Staubli VAL3: POINT.pjx

--- POINT.pjx ---
Parameters version=s7.7 stackSize=5000 millimeterUnit=true
Program file=computeFrame.pgx
Program file=delete.pgx
Program file=deleteItem.pgx
Program file=duplicate.pgx
Program file=find.pgx
Program file=get.pgx
Program file=getDistance.pgx
Program file=getFrame.pgx
Program file=getFrameId.pgx
Program file=getFunctionEdit.pgx
Program file=getFunctionSel.pgx
Program file=getFunctionView.pgx
Program file=getListItem.pgx
Program file=getPoint.pgx
Program file=getSize.pgx
Program file=getSizeItem.pgx
Program file=getTime.pgx
Program file=getTool.pgx
Program file=getTrajItem.pgx
Program file=getTrajType.pgx
Program file=getType.pgx
Program file=goTo.pgx
Program file=HerePoint.pgx
Program file=insertItem.pgx
Program file=load.pgx
Program file=loadCycle.pgx
Program file=loadPage.pgx
Program file=makeTraj.pgx
Program file=new.pgx
Program file=onEdit.pgx
Program file=onEditItem.pgx
Program file=onEditTrsf.pgx
Program file=onFunctionEdit.pgx
Program file=onFunctionSel.pgx
Program file=onFunctionView.pgx
Program file=onInsert.pgx
Program file=onProgEnd.pgx
Program file=onRun.pgx
Program file=onSave.pgx
Program file=onStart.pgx
Program file=onStop.pgx
Program file=setFrameId.pgx
Program file=setTool.pgx
Program file=setTrajItem.pgx
Data file=POINT.dtx
Library alias=saveData path=Disk://saveData/saveData.pjx
Library alias=page path=Disk://kernel/template/page/page.pjx
Library alias=use path=Disk://kernel/userPage/userPage.pjx
Library alias=language path=Disk://kernel/language/language.pjx
Library alias=tcp path=Disk://kernel/tool/tool.pjx
Library alias=cycleStatus path=Disk://cycleStatus/cycleStatus.pjx
Library alias=pt path=Disk://kernel/template/session/saveTraj/POINT/POINT.pjx
Type name=TrajectoryItem path=Disk://kernel/template/TrajectoryItem/TrajectoryItem.pjx
Type name=ActionItem path=Disk://kernel/template/ActionItem/ActionItem.pjx
Type name=Trajectory path=Disk://kernel/template/Trajectory/Trajectory.pjx
Type name=TrajPoint path=Disk://kernel/template/TrajPoint/TrajPoint.pjx
Type name=InstrItem path=Disk://kernel/template/InstrItem/InstrItem.pjx
Type name=FrameItem path=Disk://kernel/template/FrameItem/FrameItem.pjx
Type name=TrajPointItem path=Disk://kernel/template/TrajPointItem/TrajPointItem.pjx

--- POINT.dtx ---
Trajectory tTraj
  [0]
    TrajectoryItem tSuper[3]
      [0]
        num distance
        num moveType = 1
        num nTime
        num nStop
        num nTcpAction
        string comment = "appro"
        bool toStop
        mdesc nom_speed = {tmax=300, rmax=9999, leave=30, reach=30}
        InstrItem iInstr[3]
          [0]
            string sType
            string sData
          [1]
            string sType
            string sData
          [2]
            string sType
            string sData
        num nMoveId
      [1]
        num distance = 2
        num moveType = 1
        num nTime
        num nStop
        num nTcpAction = 2
        string comment = "point"
        bool toStop = true
        mdesc nom_speed = {tmax=300, rmax=9999, leave=30, reach=30}
        InstrItem iInstr[3]
          [0]
            string sType
            string sData
          [1]
            string sType
            string sData
          [2]
            string sType
            string sData
        num nMoveId
      [2]
        num distance
        num moveType = 1
        num nTime
        num nStop
        num nTcpAction
        string comment = "depart"
        bool toStop
        mdesc nom_speed = {tmax=300, rmax=9999, leave=30, reach=30}
        InstrItem iInstr[3]
          [0]
            string sType
            string sData
          [1]
            string sType
            string sData
          [2]
            string sType
            string sData
        num nMoveId
    string sID = "POINT pose"
    num nId
public bool bMoveType[3]
  [0] = true
  [1] = true
public bool bStepping
bool bToSave
frame fSetFrame = {fatherId=world[0]}
mdesc mMdesc = {accel=10, vel=10, decel=10, blend=off}
string sInstruction
public string sItems
string sMenu[8]
  [5] = "Duplicate"
  [7] = "New"
string sTrajType = "POINT"
pointRx pToGo = {fatherId=world[0]}
frame fFather = {fatherId=world[0]}
string sItemCycle
TrajPoint pEditPoint
  [0]
    TrajPointItem tData[3]
      [0]
        TrajectoryItem tSuper
          [0]
            num distance
            num moveType
            num nTime
            num nStop
            num nTcpAction
            string comment
            bool toStop
            mdesc nom_speed = {vel=500, tmax=500, rmax=9999, leave=30, reach=30}
            InstrItem iInstr[3]
              [0]
                string sType
                string sData
              [1]
                string sType
                string sData
              [2]
                string sType
                string sData
            num nMoveId
        pointRx pPoint = {fatherId=pEditPoint[0].fFrame[0]}
        num nType
      [1]
        TrajectoryItem tSuper
          [0]
            num distance
            num moveType
            num nTime
            num nStop
            num nTcpAction
            string comment
            bool toStop
            mdesc nom_speed = {vel=500, tmax=500, rmax=9999, leave=30, reach=30}
            InstrItem iInstr[3]
              [0]
                string sType
                string sData
              [1]
                string sType
                string sData
              [2]
                string sType
                string sData
            num nMoveId
        pointRx pPoint = {fatherId=pEditPoint[0].fFrame[0]}
        num nType
      [2]
        TrajectoryItem tSuper
          [0]
            num distance
            num moveType
            num nTime
            num nStop
            num nTcpAction
            string comment
            bool toStop
            mdesc nom_speed = {vel=500, tmax=500, rmax=9999, leave=30, reach=30}
            InstrItem iInstr[3]
              [0]
                string sType
                string sData
              [1]
                string sType
                string sData
              [2]
                string sType
                string sData
            num nMoveId
        pointRx pPoint = {fatherId=pEditPoint[0].fFrame[0]}
        num nType
    frame fFrame = {fatherId=world[0]}
    num nIndexTool
    string sID
    num nIndexFrame

--- computeFrame.pgx ---
public program computeFrame(num x_nNewFrame)
  local num i
begin
  // recompute all the point into the new frame
  for i=0 to size(pEditPoint.tData)-1
    if pEditPoint.tData[i].nType==1
      pEditPoint.tData[i].pPoint.trsf=position(pEditPoint.tData[i].pPoint,saveData:fFrameItem[x_nNewFrame].fFrame)
    endIf
  endFor
end

--- delete.pgx ---
public program delete(string x_sName (dimensions=1), num& x_nResult[] (dimensions=1))
  local string l_sItem
  local num l_nSize
begin
  //
  // delete the select trajectory
  //
  if isDefined(pt:tTraj[x_sName])
    // delete
    delete(pt:tTraj[x_sName])
    // save it
    bToSave=true
    x_nResult=0
  else
    x_nResult=-1
  endIf

end

--- deleteItem.pgx ---
public program deleteItem(num& x_nIndex (dimensions=1))
  local num i
  local string l_sItem
begin
  // delete the selected item
  if pEditPoint.tData[x_nIndex].nType!=1 and size(pEditPoint.tData)>3
    // delete all the field
    delete(pEditPoint.tData[x_nIndex])
  else
    // not possible to delete the point
    if pEditPoint.tData[x_nIndex].nType!=1
      pEditPoint.tData[x_nIndex].pPoint.trsf={0,0,0,0,0,0}
    endIf
    x_nIndex=-1
  endIf
end

--- find.pgx ---
public program find(string& x_sItem[] (dimensions=1), bool& x_bFound[] (dimensions=1))
begin
  // check if the item has been found
  x_bFound=isDefined(pt:tTraj[x_sItem])
end

--- get.pgx ---
public program get(string& x_sItem[] (dimensions=1), num x_nIndex (dimensions=1))
  local string l_sKey
  local num i
  local string l_sItem
begin
  // start from the first
  l_sKey=first(pt:tTraj)
  // search it
  while l_sKey!=""
    x_sItem=l_sKey
    l_sKey=next(pt:tTraj[l_sKey])
    if i==x_nIndex
      return
    else
      i=i+1
    endIf
  endWhile
end

--- getDistance.pgx ---
public program getDistance(tool x_tTool, num& x_nDistance[], bool x_bCycle, num x_nIndex)
  local point l_pPoint
  local num l_nValue
  local trsf l_trsfEmpty
  local point l_pActual
  local point l_pPrev
begin
  // first point
  if x_nIndex==0
    x_nDistance=10
    return
  else
    //
    // get the point
    //
    call getPoint(l_pActual,x_bCycle,x_nIndex)
    call getPoint(l_pPrev,x_bCycle,x_nIndex-1)
    if x_bCycle
      // an other one

      switch pt:tTraj[sItemCycle].tData[x_nIndex].nType
        case 0
          // appro
          x_nDistance=distance(position(l_pPrev,world),position(l_pActual,world))
        break
        case 1
          // point
          x_nDistance=distance(l_pPrev.trsf,l_trsfEmpty)
        break
        case 2
          // depart
          if pt:tTraj[sItemCycle].tData[x_nIndex-1].nType==1
            x_nDistance=distance(l_trsfEmpty,l_pActual.trsf)
          else
            x_nDistance=distance(position(l_pPrev,world),position(l_pActual,world))
          endIf
        break
      endSwitch
    else
      // an other one
      switch pEditPoint[x_nIndex].tData.nType
        case 0
          // appro
          x_nDistance=distance(position(l_pPrev,world),position(l_pActual,world))
        break
        case 1
          // point
          x_nDistance=distance(l_pPrev.trsf,l_trsfEmpty)
        break
        case 2
          // depart
          if pEditPoint[x_nIndex-1].tData.nType==1
            x_nDistance=distance(l_trsfEmpty,l_pActual.trsf)
          else
            x_nDistance=distance(position(l_pPrev,world),position(l_pActual,world))
          endIf
        break
      endSwitch
    endIf
  endIf
end

--- getFrame.pgx ---
public program getFrame(frame& x_fFrame[], bool x_bCycle)
begin
  if x_bCycle
    x_fFrame.trsf=position(pt:tTraj[sItemCycle].fFrame,world)
  else
    // update the frame
    x_fFrame.trsf=position(pEditPoint.fFrame,world)
  endIf
end

--- getFrameId.pgx ---
public program getFrameId(num& x_nFrame)
begin
  // give back the frame
  x_nFrame=pEditPoint.nIndexFrame
end

--- getFunctionSel.pgx ---
public program getFunctionSel(string& x_sName[] (dimensions=1))
  local string l_sMessage
begin
  //
  // define your message for the
  // function KEY
  //
  // NOTE is an ARRAY[0..7]
  //
  // example:
  // x_sName[1]="DEMO"
  // active the F2 button
  //
end

--- getListItem.pgx ---
public program getListItem(string& x_sItem[] (dimensions=1), num x_nIndex (dimensions=1))
  local trsf l_tTrsf
  local string l_sItem[6]
  local string l_sEvent
begin
  //
  // define the item to show in the edit page Traj
  // customize an array and copy to x_sItem...
  //
  // see other traj as example
  // 0 > appro
  // 1 > point
  // 2 > depart
  // take it
  switch pEditPoint.tData[x_nIndex].nType
    case 0
      l_sEvent="appro  "
    break
    case 1
      l_sEvent="coord  "
    break
    case 2
      l_sEvent="depart "
    break
  endSwitch
  l_tTrsf=pEditPoint.tData[x_nIndex].pPoint.trsf
  // show them
  l_sItem[0]=(l_sEvent+" X > "+toString(".2",l_tTrsf.x))
  l_sItem[1]=(l_sEvent+" Y > "+toString(".2",l_tTrsf.y))
  l_sItem[2]=(l_sEvent+" Z > "+toString(".2",l_tTrsf.z))
  l_sItem[3]=(l_sEvent+"RX > "+toString(".2",l_tTrsf.rx))
  l_sItem[4]=(l_sEvent+"RY > "+toString(".2",l_tTrsf.ry))
  l_sItem[5]=(l_sEvent+"RZ > "+toString(".2",l_tTrsf.rz))
  // look for intermediate point
  call use:stringCopy(l_sItem,x_sItem)
end

--- getPoint.pgx ---
public program getPoint(point& x_pPoint[], bool x_bCycle, num x_nIndex)
  local string l_sItem
  local num l_nSize
  local num i
  local num l_nPoint
begin
  // take
  if x_bCycle
    // in Cycle
    switch pt:tTraj[sItemCycle].tData[x_nIndex].nType
      case 0,2
        call getSizeItem(true,l_nSize)
        for i=0 to l_nSize-1
          // scan for the real point
          if pt:tTraj[sItemCycle].tData[i].nType==1
            l_nPoint=i
            i=l_nSize-1
          endIf
        endFor
        // give back
        x_pPoint=appro(pt:tTraj[sItemCycle].tData[l_nPoint].pPoint,pt:tTraj[sItemCycle].tData[x_nIndex].pPoint.trsf)
      break
      case 1
        // real point
        x_pPoint=pt:tTraj[sItemCycle].tData[x_nIndex].pPoint
      break
    endSwitch
  else
    // not in Cycle
    switch pEditPoint.tData[x_nIndex].nType
      case 0,2
        call getSizeItem(false,l_nSize)
        for i=0 to l_nSize-1
          // scan for the real point
          if pEditPoint.tData[i].nType==1
            l_nPoint=i
            i=l_nSize-1
          endIf
        endFor
        // give back
        x_pPoint=appro(pEditPoint.tData[l_nPoint].pPoint,pEditPoint.tData[x_nIndex].pPoint.trsf)
      break
      case 1
        // real point
        x_pPoint=pEditPoint.tData[x_nIndex].pPoint
      break
    endSwitch
  endIf
end

--- getSize.pgx ---
public program getSize(num& x_nSize[] (dimensions=1))
  local string l_sType
  local string l_sKey
  local num i
  local string l_sItem
  local string l_sPath
  local num l_nResult
begin
  // give back the size
  x_nSize=size(pt:tTraj)
end

--- getSizeItem.pgx ---
public program getSizeItem(bool x_bCycle, num& x_nSize)
  local string l_sType
  local string l_sKey
  local num i
begin
  //
  // get the size of the collection
  //
  if x_bCycle
    x_nSize=size(pt:tTraj[sItemCycle].tData)
  else
    x_nSize=size(pEditPoint.tData)
  endIf
end

--- getTime.pgx ---
public program getTime(num& x_nTime[], bool x_bCycle, num x_nIndex)
begin
  // get the time DATA
  if x_bCycle
    // get the time DATA
    x_nTime=pt:tTraj[sItemCycle].tData[x_nIndex].tSuper.nTime
  else
    // get the time DATA
    x_nTime=pEditPoint.tData[x_nIndex].tSuper.nTime
  endIf
end

--- getTool.pgx ---
public program getTool(num& x_nTool (dimensions=1))
begin
  // edit one
  x_nTool=pEditPoint.nIndexTool
end

--- getTrajItem.pgx ---
public program getTrajItem(TrajectoryItem& x_tTraj[] (dimensions=1), num x_nIndex (dimensions=1))
begin
  //
  // get all the FIELD
  //
  x_tTraj=pEditPoint.tData[x_nIndex].tSuper
end

--- getTrajType.pgx ---
program getTrajType(string& x_sTrajType[] (dimensions=1))
  local num l_nPos
  local string l_sPath
begin
  // get the trajType
  l_sPath=libPath()
  if find(l_sPath,sTrajType)==-1 or sTrajType==""
    do
      l_nPos=find(l_sPath,"/")
      if l_nPos==-1
        l_nPos=find(l_sPath,"\")
      endIf
      if l_nPos!=-1
        l_sPath=right(l_sPath,len(l_sPath)-l_nPos-1)
      endIf
    until l_nPos==-1
    //
    sTrajType=l_sPath
  endIf
  // return back
  x_sTrajType=sTrajType
end

--- getType.pgx ---
public program getType(num& x_nType, bool x_bCycle, num x_nIndex)
begin
  // get the point Type
  if x_bCycle
    x_nType=pt:tTraj[sItemCycle].tData[x_nIndex].nType
  else
    x_nType=pEditPoint.tData[x_nIndex].nType
  endIf
end

--- goTo.pgx ---
public program goTo(tool x_tTool, mdesc x_mDesc, num x_nMoveType, bool& x_bUnreached[], num x_nIndex)
  local point l_pTrsf
  local bool l_bInside
  local tool l_tTool
  local point l_pHere
  local string l_sMessage
  local num l_nSize
  local num i
  local mdesc l_mSpeed
  local joint l_jHere
  local joint l_jJoint
begin
  // the maximum size
  call getSizeItem(false,l_nSize)
  // get the trsf
  call getPoint(pToGo,false,x_nIndex)
  // check if the point is ok
  if pointToJoint(x_tTool,herej(),pToGo,l_jJoint)
    // step by step motion
    if x_nMoveType==0
      // or is not in range
      movej(pToGo,x_tTool,x_mDesc)
    else
      movel(pToGo,x_tTool,x_mDesc)
    endIf
  else
    // get the message point is not reachable
    call language:message(l_sMessage,-5)
    call use:type(0,12,"!!! "+l_sMessage)
  endIf
end

--- HerePoint.pgx ---
public program HerePoint(num x_nIndex)
  local tool l_tTool
  local point l_pHere
  local frame l_fFrame
  local num i
  local num l_nIndex
  local num l_nSize
  local string l_sMessage
begin
  //
  // take the point
  //
  // frame
  call getFrame(fSetFrame,false)
  // tool
  call tcp:getTool(l_tTool,pEditPoint.nIndexTool)
  // here
  l_pHere=here(l_tTool,fSetFrame)
  resetMotion()
  // check the index
  if pEditPoint.tData[x_nIndex].nType==1
    // save the trsf
    pEditPoint.tData[x_nIndex].pPoint.trsf=l_pHere.trsf
  else
    // search for the index of the point
    call getSizeItem(false,l_nSize)
    for i=0 to l_nSize-1
      if pEditPoint.tData[i].nType==1
        // save and exit
        l_nIndex=i
        i=l_nSize
      endIf
    endFor
    if pEditPoint.tData[l_nIndex].pPoint.trsf!={0,0,0,0,0,0}
      // compute the approch
      pEditPoint.tData[x_nIndex].pPoint.trsf=!pEditPoint.tData[l_nIndex].pPoint.trsf*l_pHere.trsf
    else
      // point not taught
      call language:message(l_sMessage,147)
      popUpMsg(l_sMessage)
    endIf
  endIf
  // check the moveType to save the config
  if pEditPoint.tData[x_nIndex].tSuper.moveType==0
    pEditPoint.tData[x_nIndex].pPoint.config=l_pHere.config
  else
    pEditPoint.tData[x_nIndex].pPoint.config={ssame,esame,wfree}
  endIf
  // to be save

end

--- insertItem.pgx ---
public program insertItem(num& x_nIndexCopy, num x_nIndexPaste)
  local num l_nLastType
  local point l_pPoint
  local num l_nType
begin
  //
  // use to add more elements from the typical one
  //
  // insert all the field
  //
  l_pPoint=pEditPoint.tData[x_nIndexCopy].pPoint
  l_nLastType=pEditPoint.tData[x_nIndexCopy].nType
  if l_nLastType==0
    l_nType=0
  elseIf l_nLastType==2 or l_nLastType==1
    l_nType=2
  endIf
  insert(pEditPoint.tData[x_nIndexPaste])
  // set IT - link it
  link(pEditPoint.tData[x_nIndexPaste].pPoint,pEditPoint.fFrame)
  pEditPoint.tData[x_nIndexPaste].pPoint.trsf=l_pPoint.trsf
  // set IT
  pEditPoint.tData[x_nIndexPaste].nType=l_nType
end

--- load.pgx ---
public program load(string x_sItem, num& x_nResult)
  local string l_sType
  local string l_sMessage
  local num i
begin
  // load the select trajectory..already loaded
  call getTrajType(l_sType)
  if find(pt:libPath(),saveData:sPathTraj)==-1
    pt:libLoad(saveData:sPathTraj+l_sType)
      delay(0)
    if saveData:bDebug
      ? "loading POINT..."+saveData:sPathTraj+l_sType
    endIf
  endIf
  // use the type...
  if isDefined(pt:tTraj[x_sItem])
    // link the frame and all the points
    call pt:link_all(x_sItem)
    // check if link and defined
    pEditPoint=pt:tTraj[x_sItem]
    pEditPoint.sID=x_sItem
  elseIf x_sItem!=""
    // not FOUND
    call language:message(l_sMessage,-7)
    x_nResult=-1
    popUpMsg(l_sMessage+x_sItem)
  endIf
end

--- loadCycle.pgx ---
public program loadCycle(string x_sItem, num& x_nResult[])
  local string l_sType
  local string l_sMessage
begin
  // load the select trajectory..already loaded
  call getTrajType(l_sType)
  if find(pt:libPath(),saveData:sPathTraj)==-1
    pt:libLoad(saveData:sPathTraj+l_sType)
    delay(0)
    if saveData:bDebug
      ? "loading POINT..."+saveData:sPathTraj+l_sType
    endIf
  endIf
  if isDefined(pt:tTraj[x_sItem])
    // link the frame and all the points
    call pt:link_all(x_sItem)
    sItemCycle=x_sItem
  else
    // not FOUND
    call language:message(l_sMessage,-7)
    x_nResult=-1
    cycleStatus:bToStop=true
    popUpMsg(l_sMessage+x_sItem)
  endIf
end

--- loadPage.pgx ---
program loadPage(string x_sPage, string& x_sItems[])
// load the next page
  local num i
begin
  // look if the page libload is correct
  i=page:libLoad(x_sPage)
  delay(0)
  logMsg("KERNEL:PAGE LIBLOAD "+x_sPage+" result "+toString("",i))
  if i!=0
    popUpMsg("Loading page "+x_sPage+" error CODE "+toString("",i))
  else
    page:sItems=x_sItems
    call page:main()
  endIf
end

--- makeTraj.pgx ---
public program makeTraj(string& x_sItem[])
  local num i
  local num l_nDistance
  local num l_nSize
  local tool l_tTool
  local bool l_bToStop
  local mdesc l_mDesc
  local num l_nMoveId
  local bool l_bOk
  local string l_sType
  local TrajectoryItem l_tTraj
  local ActionItem l_aAction
  local point l_pPoint
begin
  // take the TOOL
  call tcp:getTool(l_tTool,pt:tTraj[sItemCycle].nIndexTool)
  // the maximum size
  call getSizeItem(true,l_nSize)
  //
  // for all of my traj cyclePoints move the robot
  //
  resize(tTraj.tSuper,1,size(pt:tTraj[sItemCycle].tData))
  for i=0 to (l_nSize-1)
    tTraj.tSuper[i]=pt:tTraj[sItemCycle].tData[i].tSuper
  endFor
  tTraj.sID="POINT "+pt:tTraj[sItemCycle].sID
  call cycleStatus:addTraj(tTraj)
  //
  // for all of my traj cyclePoints move the robot
  //
  for i=0 to (l_nSize-1)
    //
    // get the point info
    //
    l_tTraj=pt:tTraj[sItemCycle].tData[i].tSuper
    call getPoint(l_pPoint,true,i)
    //
    // get the distance in percentage
    call getDistance(l_tTool,l_nDistance,true,i)
    //
    // give to the traj library the percentage distance
    //
    if l_bToStop
      l_tTraj.nom_speed.blend=off
    endIf
    //
    // put the move in the stack
    //
    switch pt:tTraj[sItemCycle].tData[i].nType
      case 0
        // check if the next point is the reference point
        if !(pt:tTraj[sItemCycle].tData[i+1].nType==1 and pt:tTraj[sItemCycle].tData[i].pPoint.trsf=={0,0,0,0,0,0})
          // approach
          if l_tTraj.moveType==0
            // or is not in range
            l_nMoveId=movej(l_pPoint,l_tTool,l_tTraj.nom_speed)
          else
            l_nMoveId=movel(l_pPoint,l_tTool,l_tTraj.nom_speed)
          endIf
        else
          // set as the last MOVEID
          call cycleStatus:getLastId(l_nMoveId)
          // check the index
          if i==0
            l_nMoveId=l_nMoveId+1
          endIf
        endIf
      break
      case 1
        //point
        if l_tTraj.moveType==0
          // or is not in range
          l_nMoveId=movej(l_pPoint,l_tTool,l_tTraj.nom_speed)
        else
          l_nMoveId=movel(l_pPoint,l_tTool,l_tTraj.nom_speed)
        endIf
      break
      case 2
        //  depart
        // check if the next point is the reference point
        if !(pt:tTraj[sItemCycle].tData[i-1].nType==1 and pt:tTraj[sItemCycle].tData[i].pPoint.trsf=={0,0,0,0,0,0})
          if l_tTraj.moveType==0
            // or is not in range
            l_nMoveId=movej(l_pPoint,l_tTool,l_tTraj.nom_speed)
          else
            l_nMoveId=movel(l_pPoint,l_tTool,l_tTraj.nom_speed)
          endIf
        else
          // set as the last MOVEID
          call cycleStatus:getLastId(l_nMoveId)
        endIf
      break
    endSwitch
    //
    // set the ID
    //
    l_aAction.nDistance=l_nDistance
    l_aAction.nPointId=i
    l_aAction.nMoveId=l_nMoveId
    l_aAction.sIdTraj="POINT "+pt:tTraj[sItemCycle].sID
    call cycleStatus:putInstr_Traj(l_aAction,l_tTraj,pt:tTraj[sItemCycle].nIndexTool,l_nSize)
    // there is a waitEndMove
    if l_tTraj.toStop
      waitEndMove()
      delay(l_tTraj.nStop)
      // wait all the action has been done
      wait(cycleStatus:bActionRunning==false)
    endIf
  endFor
  // bye bye
end

--- new.pgx ---
public program new(string x_sName (dimensions=1), num& x_nResult[] (dimensions=1))
  local string l_sPrefix
  local num l_nResult
begin
  // new one
  if insert(pt:tTraj[x_sName])
    call pt:link_it(x_sName)
    pt:tTraj[x_sName].nIndexTool=saveData:nIndexTool
    x_nResult=0
    // set it
    bToSave=true
  else
    x_nResult=-1
  endIf
end

--- onEdit.pgx ---
public program onEdit(string& x_sItem[])
  local string l_sPath
  local num i
  local string l_sItem
  local num l_nSize
  local num l_nResult
begin
  // DEFINE YOUR ITEM
  call getTrajType(saveData:sTrajTypeUsing)
  // load the trajectory
  call load(x_sItem,l_nResult)
  if find(x_sItem,"@")==-1
    // load the page viewTraj
    l_sPath="Disk://trajectory/page_viewTraj"
    // give back the path
    x_sItem[1]=x_sItem
    x_sItem=l_sPath
  endIf
end

--- onEditItem.pgx ---
public program onEditItem(string& x_sEvent[] (dimensions=1), num x_nIndex (dimensions=1), num x_nIndexItem (dimensions=1))
begin
  // edit the custom element that was add in the list
  call onEditTrsf(x_nIndex,x_nIndexItem,x_sEvent)
end

--- onEditTrsf.pgx ---
public program onEditTrsf(num x_nIndex (dimensions=1), num x_nIndexItem (dimensions=1), string x_sEvent (dimensions=1))
  local num i
  local num l_nMin
  local num l_nMax
  local trsf l_tTrsf
  local string l_sEmpty
begin
  // edit TRSF OF THE POINT
  l_tTrsf=pEditPoint.tData[x_nIndexItem].pPoint.trsf
  // find the >
  call use:findPos(x_sEvent,">",i)
  i=i+1
  // find the line
  if !cycleStatus:bCycle
    l_nMin=l_nMax=0
  else
    switch x_nIndex
      case 0
        // x
        l_nMin=l_tTrsf.x-10
        l_nMax=l_tTrsf.x+10
      break
      case 1
        // y
        l_nMin=l_tTrsf.y-10
        l_nMax=l_tTrsf.y+10
      break
      case 2
        // z
        l_nMin=l_tTrsf.z-10
        l_nMax=l_tTrsf.z+10
      break
      case 3
        // rx
        l_nMin=l_tTrsf.rx-5
        l_nMax=l_tTrsf.rx+5
      break
      case 4
        // ry
        l_nMin=l_tTrsf.ry-5
        l_nMax=l_tTrsf.ry+5
      break
      case 5
        // rz
        l_nMin=l_tTrsf.rz-5
        l_nMax=l_tTrsf.rz+5
      break
    endSwitch
  endIf
  // clean the line
  call use:listcursor(use:nView,false)
  //
  switch x_nIndex
    case 0
      //  x-value
      call use:changeValue(l_tTrsf.x,l_nMin,l_nMax,i+40-use:nBottomX,use:nView+1,l_sEmpty)
    break
    case 1
      //  y-value
      call use:changeValue(l_tTrsf.y,l_nMin,l_nMax,i+40-use:nBottomX,use:nView+1,l_sEmpty)
    break
    case 2
      //  z-value
      call use:changeValue(l_tTrsf.z,l_nMin,l_nMax,i+40-use:nBottomX,use:nView+1,l_sEmpty)
    break
    case 3
      //  rx-value
      call use:changeValue(l_tTrsf.rx,l_nMin,l_nMax,i+40-use:nBottomX,use:nView+1,l_sEmpty)
    break
    case 4
      //  ry-value
      call use:changeValue(l_tTrsf.ry,l_nMin,l_nMax,i+40-use:nBottomX,use:nView+1,l_sEmpty)
    break
    case 5
      //  rz-value
      call use:changeValue(l_tTrsf.rz,l_nMin,l_nMax,i+40-use:nBottomX,use:nView+1,l_sEmpty)
    break
  endSwitch
  // validate
  if !use:bUseEscape
    pEditPoint.tData[x_nIndexItem].pPoint.trsf=l_tTrsf
  endIf
end

--- onFunctionEdit.pgx ---
public program onFunctionEdit(num x_nIndex, string x_sEvent, num x_nFunctionKey)
  local string l_sMessage
  local string l_sButton[2]
  local bool l_bOk
  local string l_sPage
  local string l_sItem
  local tool l_tTool
  local point l_pAlign
  local bool l_bYes
  local string l_sMessage2
  local joint l_jJoint
begin
  //
  // do on Key action
  //
  // x_nIndex = actual index item
  // x_sEvent = actual event item
  //
  switch x_nFunctionKey
    // F1 button
    case 271
      // HERE JOINT
      if !cycleStatus:bCycle
        call language:message(l_sMessage,160)
        call language:getYesNo(l_sButton)
        call use:yes_no(l_sMessage,l_sButton,l_bYes)
        if l_bYes
          call HerePoint(x_nIndex)
        endIf
      endIf
    break
    // F2 button
    case 272
      // ALIGN
      if !cycleStatus:bCycle
        resetMotion()
        call getFrame(fSetFrame,false)
        // tool
        call tcp:getTool(l_tTool,pEditPoint.nIndexTool)
        l_pAlign=here(l_tTool,world)
        l_pAlign.trsf=align(l_pAlign.trsf,fSetFrame.trsf)
        if pointToJoint(l_tTool,herej(),l_pAlign,l_jJoint)
          call language:message(l_sMessage,203)
          call language:message(l_sMessage2,134)
          l_sMessage=l_sMessage+" "+l_sMessage2+"..."
          call use:timerDialog(l_sMessage,0)
          movej(l_pAlign,l_tTool,mMdesc)
          watch(isEmpty() or isKeyPressed(255),3)
          delay(2)
        endIf
      endIf
    break
    // F3 button
    case 273

    break
    // F4 button
    case 274
    break
    // F5 button
    case 275
    break
    // F6 button
    case 276
    break
    // F7 button
    case 277
    break
    // F8 button
    case 278
      // save it
      bToSave=true
    break
  endSwitch
end

--- onFunctionSel.pgx ---
public program onFunctionSel(num x_nIndex (dimensions=1), string x_sEvent (dimensions=1), num x_nFunctionKey (dimensions=1))
begin
  //
  // do on Key action
  //
  // x_nIndex = actual index item
  // x_sEvent = actual event item
  //
  switch x_nFunctionKey
    // F1 button
    case 271
    break
    // F2 button
    case 272
    break
    // F3 button
    case 273
    break
    // F4 button
    case 274
    break
    // F5 button
    case 275
    break
    // F6 button
    case 276
    break
    // F7 button
    case 277
    break
    // F8 button
    case 278
    break
  endSwitch
end

--- onFunctionView.pgx ---
public program onFunctionView(num x_nIndex, string x_sEvent, num x_nFunctionKey)
  local string l_sMessage
  local string l_sPage
  local string l_sItem
  local string l_sButton[2]
  local bool l_bYes
  local tool l_tTool
  local point l_pAlign
  local string l_sMessage2
  local joint l_jJoint
begin
  //
  // do on Key action
  //
  // x_nIndex = actual index item
  // x_sEvent = actual event item
  //
  switch x_nFunctionKey
    // F1 button
    case 271
      // HERE JOINT
      if !cycleStatus:bCycle
        call language:message(l_sMessage,160)
        call language:getYesNo(l_sButton)
        call use:yes_no(l_sMessage,l_sButton,l_bYes)
        if l_bYes
          call HerePoint(x_nIndex)
        endIf
      endIf
    break
    // F2 button
    case 272
      // ALIGN
      if !cycleStatus:bCycle and !cycleStatus:bSimulation
        resetMotion()
        call getFrame(fSetFrame,false)
        // tool
        call tcp:getTool(l_tTool,pEditPoint.nIndexTool)
        l_pAlign=here(l_tTool,world)
        l_pAlign.trsf=align(l_pAlign.trsf,fSetFrame.trsf)
        // check the align
        if pointToJoint(l_tTool,herej(),l_pAlign,l_jJoint)
          call language:message(l_sMessage,203)
          call language:message(l_sMessage2,134)
          l_sMessage=l_sMessage+" "+l_sMessage2+"..."
          call use:timerDialog(l_sMessage,0)
          movej(l_pAlign,l_tTool,mMdesc)
          watch(isEmpty() or isKeyPressed(255),3)
          if !isEmpty()
            resetMotion()
          endIf
          delay(2)
        endIf
      endIf
    break
    // F3 button
    case 273
    break
    // F4 button
    case 274
    break
    // F5 button
    case 275
    break
    // F6 button
    case 276
    break
    // F7 button
    case 277
    break
    // F8 button
    case 278
    break
  endSwitch
end

--- onInsert.pgx ---
public program onInsert(string& x_sItem[] (dimensions=1))
  local string l_sEvent
  local num l_nKey
  local num l_nIndex
  local num l_nSize
  local num i
  local string l_sMessage
  local bool l_bFound
  local string l_sType
  local bool l_bUseFilter
  local string l_sPaste
  local num l_nResult
  local num l_nX
  local num l_nY
  local string l_sName
begin
  // get the type
  call getTrajType(x_sItem)
  saveData:sTrajTypeUsing=x_sItem
  cls()
  // is a filter using ??
  if saveData:sTrajFilter!=""
    l_bUseFilter=true
    call language:message(l_sMessage,64)
    call use:type(0,1,l_sMessage+">ON")
  else
    // clean
    call use:typeLen(0,1," ",use:nBottomX)
  endIf
  //
  // CREATE THE LIST
  //
  // define your list size for default
  call use:setSizeList(19,0,19,11)
  call use:setView(false)
  call use:listcreate(x_sItem)
  // take the coordinate....
  l_nX=40-use:nBottomX-1
  l_nY=use:nBottomY+1
  // show the message
  call language:message(l_sMessage,61)
  call use:stringToArray(l_sMessage,sMenu)
  call use:setMenu(sMenu,true,3)
  // Build the list
  call getSize(l_nSize)
  for i=0 to l_nSize-1
    call get(l_sEvent,i)
    if l_sEvent!=""
      //
      // use the filter ?
      //
      // check if the bProcessList filter is active
      //
      l_bFound=true
      if saveData:sTrajFilter!=""
        l_bFound=find(l_sEvent,saveData:sTrajFilter)!=-1
      endIf
      // add
      if l_bFound
        call use:listadd(l_sEvent)
      endIf
    endIf
  endFor
  call use:listupdate(0)
  do
    // get the item
    l_nKey=get()
    call use:listevent(l_nKey,l_nIndex,l_sEvent)
    if l_nKey==271 and l_bUseFilter
      // Build the list
      call getSize(l_nSize)
      // empty and rebuild
      call use:listempty()
      for i=0 to l_nSize-1
        call get(l_sEvent,i)
        if l_sEvent!=""
          call use:listadd(l_sEvent)
        endIf
      endFor
      // clean
      call use:typeLen(0,1," ",use:nBottomX)
      call use:typeMenu(1," ")
      l_bUseFilter=false
      call use:listupdate(0)
    endIf
    //
  until l_nKey==270 or l_nKey==255 or l_nKey==278 or l_nKey==276
  //
  switch l_nKey
    case 270
      // save the name
      l_sName=l_sEvent
    break
    case 276
      // duplicate
      // ask for the new
      call language:message(l_sMessage,21)
      call use:type(l_nX,l_nY,l_sMessage)
      l_sName=l_sEvent
      // read the new trajectory
      call use:read(l_nX+len(l_sMessage),l_nY,l_sName,10,false)
      if !use:bUseEscape
        call duplicate(l_sEvent,l_sName,l_nResult)
      endIf
    break
    case 278
      call language:message(l_sMessage,21)
      call use:type(l_nX,l_nY,l_sMessage)
      // read the new trajectory
      call use:read(l_nX+len(l_sMessage),l_nY,l_sName,10,false)
      if !use:bUseEscape
        // look if the items exist
        call new(l_sName,l_nResult)
        if l_nResult==-1
          call language:message(l_sMessage,-2)
          popUpMsg(l_sMessage)
        endIf
      endIf
    break
  endSwitch
  if l_nKey!=255
    x_sItem=l_sName
  else
    x_sItem=""
  endIf
end

--- onProgEnd.pgx ---
public program onProgEnd(string& x_sItem[] (dimensions=1))
begin
end

--- onRun.pgx ---
public program onRun(string& x_sItem[] (dimensions=1))
  local string l_sEmpty
  local num l_nResult
begin
  // execute check if need to reload
  call loadCycle(x_sItem,l_nResult)
  // execute
  call makeTraj(x_sItem)
end

--- onSave.pgx ---
public program onSave(string& x_sItem[])
  local num i
  local num l_nSize
begin
  //if bToSave
  // update
  if isDefined(pt:tTraj[pEditPoint.sID])
    pt:tTraj[pEditPoint.sID]=pEditPoint
    // loink all the point
    call pt:link_all(pEditPoint.sID)
  endIf
  // saveIt
  pt:libSave()
  bToSave=false
  // endIf
end

--- onStart.pgx ---
public program onStart(string& x_sItem[] (dimensions=1))
  local num i
  local string l_sType
begin

end

--- onStop.pgx ---
public program onStop(string& x_sItem[])
begin
  // stop it
  if x_sItem=="kill"
    pt:libLoad("Disk://kernel/template/session/saveTraj/POINT")
  endIf
end

--- setFrameId.pgx ---
public program setFrameId(num x_nIndex)
  local num i
begin
  //
  // save the FrameId
  //
  pEditPoint.nIndexFrame=x_nIndex
  // link to the father frame and alll the point
  link(pEditPoint.fFrame,saveData:fFrameItem[x_nIndex].fFrame)
  for i=0 to size(pEditPoint.tData)-1
    link(pEditPoint.tData[i].pPoint,pEditPoint.fFrame)
  endFor
end

--- setTool.pgx ---
public program setTool(num x_nIndexTool (dimensions=1))
begin
  // set the TOOL
  pEditPoint.nIndexTool=x_nIndexTool
end

--- setTrajItem.pgx ---
public program setTrajItem(TrajectoryItem& x_tTraj[] (dimensions=1), num x_nIndex (dimensions=1))
begin
  //
  // set all the field
  //
  pEditPoint.tData[x_nIndex].tSuper=x_tTraj
  // active the save data
  bToSave=true
end
